(* CODESYS project Untitled1.project

Project tree, tasks and I/O mapping:
  Device : CODESYS Control Win V3, 3S - Smart Software Solutions GmbH, order no. 305021, version 3.5.11.30
    application Application
      libraries: Standard, * (System)
      task MainTask (cyclic, interval t#20ms, priority 1) calls PLC_PRG
      program PLC_PRG [SFC]: P1_active, P3_active, P4_active, P5_active, P6_active, P7_active, P8_active, P9_active, P10_active, P11_active, P0_active, P12_active, P13_active, P14_active, P2_active, P15_active, P16_active, P17_active, P18_active, P25_active
*)

// Device/Application/PLC_PRG
PROGRAM PLC_PRG
VAR
	BTA: BOOL;
	AUTO: BOOL;
	BTM: BOOL;
	C1: BOOL;
	M2_2: BOOL;
	B: BOOL;
	IM1: BOOL;
	M2_1: BOOL;
	A: BOOL;
	M1_1: BOOL;
	C2: BOOL;
	C3: BOOL;
	M1_2: BOOL;
	B1: BOOL;
	B2: BOOL;
	B3: BOOL;
	B4: BOOL;
	B5: BOOL;
	MAN: BOOL;
	BTS: BOOL;
	R1: R_TRIG;
	CONT: INT;
	RESET: BOOL;
END_VAR

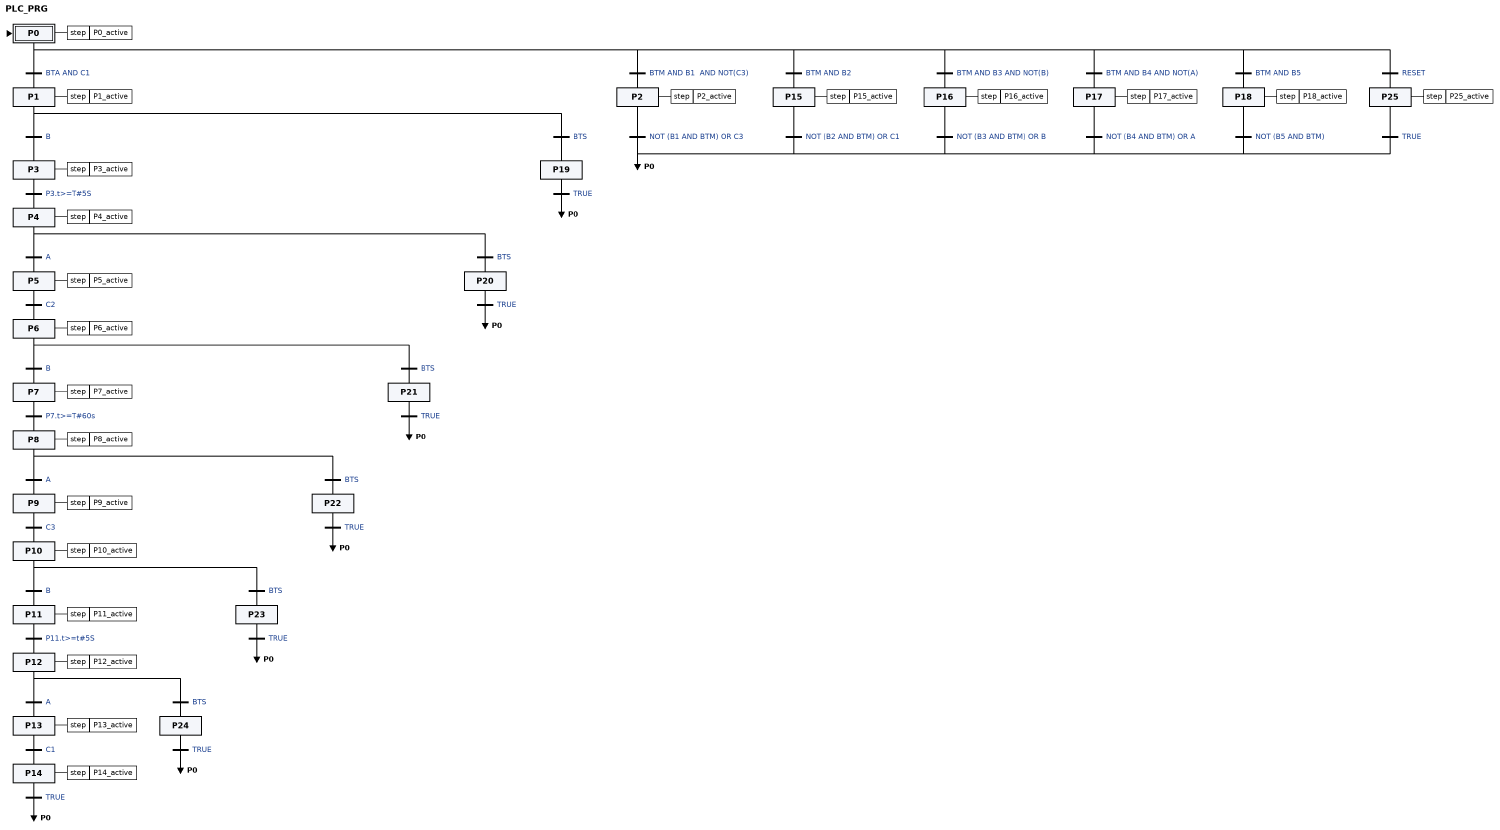
INITIAL_STEP P0:
    P0_active(N);  // step action
END_STEP
TRANSITION FROM P0 TO P1
    := BTA AND C1;
END_TRANSITION
STEP P1:
    P1_active(N);  // step action
END_STEP
TRANSITION FROM P1 TO P3
    := B;
END_TRANSITION
STEP P3:
    P3_active(N);  // step action
END_STEP
TRANSITION FROM P3 TO P4
    := P3.t>=T#5S;
END_TRANSITION
TRANSITION FROM P1 TO P19
    := BTS;
END_TRANSITION
STEP P19:
END_STEP
TRANSITION FROM P19 TO P0
    := TRUE;
END_TRANSITION
STEP P4:
    P4_active(N);  // step action
END_STEP
TRANSITION FROM P4 TO P5
    := A;
END_TRANSITION
STEP P5:
    P5_active(N);  // step action
END_STEP
TRANSITION FROM P5 TO P6
    := C2;
END_TRANSITION
TRANSITION FROM P4 TO P20
    := BTS;
END_TRANSITION
STEP P20:
END_STEP
TRANSITION FROM P20 TO P0
    := TRUE;
END_TRANSITION
STEP P6:
    P6_active(N);  // step action
END_STEP
TRANSITION FROM P6 TO P7
    := B;
END_TRANSITION
STEP P7:
    P7_active(N);  // step action
END_STEP
TRANSITION FROM P7 TO P8
    := P7.t>=T#60s;
END_TRANSITION
TRANSITION FROM P6 TO P21
    := BTS;
END_TRANSITION
STEP P21:
END_STEP
TRANSITION FROM P21 TO P0
    := TRUE;
END_TRANSITION
STEP P8:
    P8_active(N);  // step action
END_STEP
TRANSITION FROM P8 TO P9
    := A;
END_TRANSITION
STEP P9:
    P9_active(N);  // step action
END_STEP
TRANSITION FROM P9 TO P10
    := C3;
END_TRANSITION
TRANSITION FROM P8 TO P22
    := BTS;
END_TRANSITION
STEP P22:
END_STEP
TRANSITION FROM P22 TO P0
    := TRUE;
END_TRANSITION
STEP P10:
    P10_active(N);  // step action
END_STEP
TRANSITION FROM P10 TO P11
    := B;
END_TRANSITION
STEP P11:
    P11_active(N);  // step action
END_STEP
TRANSITION FROM P11 TO P12
    := P11.t>=t#5S;
END_TRANSITION
TRANSITION FROM P10 TO P23
    := BTS;
END_TRANSITION
STEP P23:
END_STEP
TRANSITION FROM P23 TO P0
    := TRUE;
END_TRANSITION
STEP P12:
    P12_active(N);  // step action
END_STEP
TRANSITION FROM P12 TO P13
    := A;
END_TRANSITION
STEP P13:
    P13_active(N);  // step action
END_STEP
TRANSITION FROM P13 TO P14
    := C1;
END_TRANSITION
TRANSITION FROM P12 TO P24
    := BTS;
END_TRANSITION
STEP P24:
END_STEP
TRANSITION FROM P24 TO P0
    := TRUE;
END_TRANSITION
STEP P14:
    P14_active(N);  // step action
END_STEP
TRANSITION FROM P14 TO P0
    := TRUE;
END_TRANSITION
TRANSITION FROM P0 TO P2
    := BTM AND B1 AND NOT(C3);
END_TRANSITION
STEP P2:
    P2_active(N);  // step action
END_STEP
TRANSITION FROM P2 TO P0
    := NOT (B1 AND BTM) OR C3;
END_TRANSITION
TRANSITION FROM P0 TO P15
    := BTM AND B2;
END_TRANSITION
STEP P15:
    P15_active(N);  // step action
END_STEP
TRANSITION FROM P15 TO P0
    := NOT (B2 AND BTM) OR C1;
END_TRANSITION
TRANSITION FROM P0 TO P16
    := BTM AND B3 AND NOT(B);
END_TRANSITION
STEP P16:
    P16_active(N);  // step action
END_STEP
TRANSITION FROM P16 TO P0
    := NOT (B3 AND BTM) OR B;
END_TRANSITION
TRANSITION FROM P0 TO P17
    := BTM AND B4 AND NOT(A);
END_TRANSITION
STEP P17:
    P17_active(N);  // step action
END_STEP
TRANSITION FROM P17 TO P0
    := NOT (B4 AND BTM) OR A;
END_TRANSITION
TRANSITION FROM P0 TO P18
    := BTM AND B5;
END_TRANSITION
STEP P18:
    P18_active(N);  // step action
END_STEP
TRANSITION FROM P18 TO P0
    := NOT (B5 AND BTM);
END_TRANSITION
TRANSITION FROM P0 TO P25
    := RESET;
END_TRANSITION
STEP P25:
    P25_active(N);  // step action
END_STEP
TRANSITION FROM P25 TO P0
    := TRUE;
END_TRANSITION

ACTION P1_active:
M2_2 := TRUE;
AUTO:=TRUE;
END_ACTION

ACTION P3_active:
IM1:=TRUE;
M2_2 := FALSE;
END_ACTION

ACTION P4_active:
M2_1:=TRUE;
END_ACTION

ACTION P5_active:
M2_1:=FALSE;
M1_1:=TRUE;
END_ACTION

ACTION P6_active:
M1_1:=FALSE;
M2_2:= TRUE;
END_ACTION

ACTION P7_active:
R1(CLK:=B);
IF R1.Q THEN 
	CONT := CONT+1;
END_IF
M2_2:= FALSE;
END_ACTION

ACTION P8_active:
M2_1:=TRUE;
END_ACTION

ACTION P9_active:
M2_1:=FALSE;
M1_1:=TRUE;
END_ACTION

ACTION P10_active:
M1_1:=FALSE;
M2_2:=TRUE;
END_ACTION

ACTION P11_active:
M2_2:=FALSE;
IM1:=FALSE;
END_ACTION

ACTION P0_active:
AUTO:=FALSE;
MAN:=FALSE;
M1_1:=FALSE;
M1_2:=FALSE;
M2_2:=FALSE;
M2_1:=FALSE;
IM1:=FALSE;
END_ACTION

ACTION P12_active:
M2_1:=TRUE;
END_ACTION

ACTION P13_active:
M2_1:=FALSE;
M1_2:=TRUE;
END_ACTION

ACTION P14_active:
M1_2:=FALSE;
END_ACTION

ACTION P2_active:
MAN:=TRUE;
M1_1:=TRUE;
END_ACTION

ACTION P15_active:
M1_2:=TRUE;
MAN:= TRUE;
END_ACTION

ACTION P16_active:
MAN := TRUE;
M2_2 :=TRUE;
END_ACTION

ACTION P17_active:
MAN:= TRUE;
M2_1:=TRUE;
END_ACTION

ACTION P18_active:
MAN:= TRUE;
IM1:=TRUE;
END_ACTION

ACTION P25_active:
CONT:=0;
END_ACTION

END_PROGRAM
